{attribute 'GeneratedUsingTerminal: EP2316-0008-0016'}
{attribute addProperty BoxType "EP2316-0008-0016"}
{attribute addProperty Id "Safe_state_activeAT %I*BOOL1Error_channel_1AT %I*BOOL1Sync_ErrorAT %I*BOOL1TxPDO_ToggleAT %I*BOOL1"}
{attribute addProperty CRC "2937461406"}
{attribute addProperty Size "4"}
TYPE DO_Inputs_Device_AF161A9E :
STRUCT
	{attribute addProperty Name "Safe_state_active"}
	Safe_state_active AT %I* : BOOL;
	{attribute addProperty Name "Error_channel_1"}
	Error_channel_1 AT %I* : BOOL;
	{attribute addProperty Name "Sync_Error"}
	Sync_Error AT %I* : BOOL;
	{attribute addProperty Name "TxPDO_Toggle"}
	TxPDO_Toggle AT %I* : BOOL;
END_STRUCT
END_TYPE

(* stored: Version 1.2.0.0, ProductVersion 3.1.4024.9
   DUT DO_Inputs_Device_AF161A9E: Id {7e2a46c3-fafb-426b-b03f-fe4f379feb4b} *)
